TYPE Room_Settings_TempTime :
STRUCT
	timee	: Room_Settings_TimeSettings;
	temp	: Room_Settings_TemperatureSettings;
END_STRUCT
END_TYPE

(* stored: Version 1.1.0.1
   DUT Room_Settings_TempTime: Id {79dbd6a5-e9a2-4b6b-8eee-c25dee1a2934} *)
